VAR_GLOBAL
// B940-008-L0S23-PNL-1 (Fee)
{attribute 'pytmc' := ' pv: TXI:ST1L1:GCC:01 '}
fb_ST1L1_GCC_01: FB_MKS500;
{attribute 'pytmc' := ' pv: TXI:ST1L1:GPI:01 '}
fb_ST1L1_GPI_01: FB_MKS275;


// B950-100H1-L1S1-PNL-1 (H1.1)
{attribute 'pytmc' := ' pv: TXI:TV3L1_GCC:01 '}
fb_TV3L1_GCC_01: FB_MKS500;
{attribute: 'pytmc' := ' pv: TXI:TV3l1:GPI:01 '}
fb_TV3L1_GPI_01: FB_MKS275;

// B950-100H1-L1S3-DRL-1 (H1.1)
{attribute: 'pytmc' := 'pv: TXI:TV5L1-GCC:01 '}
fb_TV5L1_GCC_01: FB_MKS500;
{attribute: 'pytmc' := ' pv: TXI:TV5L1:GPI:01 '}
fb_TV5L1_GPI_01: FB_MKS275;
END_VAR

(* stored: Version 1.1.0.1, ProductVersion 3.1.4024.6
   GVL GVL_TXI_VAC_GAUGES: Id {716e6ff7-4b20-47dc-ba4c-6ff2f55b9074} *)
